FUNCTION_BLOCK ButtonNC EXTENDS Button
VAR
	input AT %I* : BOOL;
END_VAR

PROPERTY IsPressed : BOOL
GET
IsPressed := NOT input;
END_GET
END_PROPERTY

PROPERTY IsReleased : BOOL
GET
IsReleased := input;
END_GET
END_PROPERTY

END_FUNCTION_BLOCK

(* stored: Version 1.1.0.1, ProductVersion 3.1.4024.12
   POU ButtonNC: Id {3e3211aa-f658-4283-830b-d1464a00a171}, SpecialFunc None
   Property IsPressed: Id {8ca30260-2150-4264-8ab6-f1ec95f60bc3}
   Get Get: Id {b9e1107d-adf6-4b28-a350-8cb0ca0076fb}
   Property IsReleased: Id {009371a7-3770-477f-ad31-4edbccc7be49}
   Get Get: Id {41573aa6-e79b-4204-89cf-62dae66aac19} *)
